// TIA Portal V17 export
// export: Created 2025-03-05T08:02:23.0636914Z, ExportSetting WithDefaults, DisplayName Totally Integrated Automation Portal, DisplayVersion V17 Update 8, DisplayName TIA Portal Openness, DisplayVersion V17 Update 8, DisplayName TIA Portal Version Control Interface, DisplayVersion V17, DisplayName SINAMICS Startdrive Advanced, DisplayVersion V17 SP2, DisplayName SINAMICS Startdrive G110M, G120, G120C, G120D, G120P, G115D, DisplayVersion V17 SP2, DisplayName SINAMICS Startdrive G130, G150, S120, S150, SINAMICS MV, S210, DisplayVersion V17 SP2, DisplayName STEP 7 Professional, DisplayVersion V17 Update 8, DisplayName SINUMERIK ONE STEP 7 Toolbox, DisplayVersion V17 Update 12, DisplayName SINUMERIK 840D sl STEP 7 Toolbox, DisplayVersion V17 Update 12, DisplayName STEP 7 Safety, DisplayVersion V17 Update 6, DisplayName WinCC Advanced, DisplayVersion V17 Update 8
TYPE "SAFETY_DOOR"
// stored: IsFailsafeCompliant false
   STRUCT
      CLOSED_I : Bool;   // CLOSED INPUT
      LOCKED_I : Bool;   // LOCKED INPUT
      OPEN_I : Bool;   // OPENED INPUT / OPEN INPUT
      UNLOCKED_I : Bool;   // UNLOCKED INPUT
      LOCK_GENERAL_CONDITIONS : Bool;   // LOCK GENERAL CONDITIONS
      LOCK_MANUAL_REQUEST : Bool;   // LOCK MANUAL REQUEST
      LOCK_HMI_REQUEST : Bool;   // LOCK SAFETY DOOR HMI REQUEST / LOCK HMI REQUEST
      LOCK_AUTO_REQUEST : Bool;   // LOCK AUTO REQUEST
      LOCK_GLOBAL_REQUEST : Bool;   // LOCK GLOBAL REQUEST
      LOCK_COMMAND : Bool;   // LOCK COMMAND
      LOCK : Bool;   // LOCK
      CLOSED_AND_LOCKED : Bool;   // CLOSED AND LOCKED
      UNLOCK_GENERAL_CONDITIONS : Bool;   // UNLOCK GENERAL CONDITIONS
      PARTIAL_UNLOCK_GENERAL_CONDITIONS : Bool;   // PARTIAL UNLOCK GENERAL CONDITIONS
      UNLOCK_MANUAL_REQUEST : Bool;   // UNLOCK MANUAL REQUEST
      UNLOCK_HMI_REQUEST : Bool;   // UNLOCK SAFETY DOOR HMI REQ / UNLOCK HMI REQUEST
      UNLOCK_AUTO_REQUEST : Bool;   // UNLOCK AUTO REQUEST
      UNLOCK_GLOBAL_REQUEST : Bool;   // UNLOCK GLOBAL REQUEST
      UNLOCK_COMMAND : Bool;   // UNLOCK COMMAND
      UNLOCK : Bool;   // UNLOCK
      OPEN_OR_UNLOCKED : Bool;   // OPENED AND UNLOCKED / OPEN OR UNLOCKED
      NOT_CLOSED_AND_LOCKED_ALARM : Bool;   // SAFETY DOOR FAULT / NOT CLOSED AND LOCKED ALARM
      DEPRESSURIZE_HYDRAULIC_DRIVE_ALARM : Bool;   // NOT POSSIBLE TO UNLOCK DEPRESSURIZE HYDRAULIC DRIVE ALARM
      NOT_CLOSED_AND_LOCKED_PREALARM : Bool;   // SAFE DOOR NOT CLOSED HELP / NOT CLOSED AND LOCKED WARNING
      UNLOCK_REQUEST_WARNING : Bool;   // UNLOCK REQUEST WARNING
      LOCK_GENERAL_CONDITIONS_HELP : Bool;   // LOCK GENERAL CONDITIONS HELP
      UNLOCK_GENERAL_CONDITIONS_HELP : Bool;   // UNLOCK GENERAL CONDITIONS HELP
      LOCK_MANUAL_REQUEST_AUX : Bool;   // AUXILIAR UNLOCK / LOCK MANUAL REQUEST AUXILIARY
      PARTIAL_UNLOCK_GENERAL_CONDITIONS_AUX : Bool;   // AUXILIAR UNLOCK / PARTIAL UNLOCK GENERAL CONDITIONS AUXILIARY
      UNLOCK_MANUAL_REQUEST_AUX : Bool;   // AUXILIAR UNLOCK / UNLOCK MANUAL REQUEST AUXILIARY
      UNLOCK_AUTO_REQUEST_AUX : Bool;   // AUXILIAR UNLOCK / UNLOCK AUTO REQUEST AUXILIARY
      UNLOCK_AUX : Bool;   // AUXILIAR UNLOCK / UNLOCK AUXILIARY
      PREALARM_GONE : Bool;   // AUXILIAR UNLOCK / WARNING GONE
      TIMER_PARTIAL_UNLOCK_GENERAL_CONDITIONS : TON_TIME;   // PARTIAL UNLOCK GENERAL CONDITIONS TIMER
      TIMER_UNLOCK : TON_TIME;   // UNLOCK TIMER
      TIMER_NOT_POSSIBLE_TO_UNLOCK : TON_TIME;   // NOT POSSIBLE TO UNLOCK TIMER
   END_STRUCT;
END_TYPE
